{attribute 'pack_mode' := '1'}
TYPE ST_ReportListItem_Test :
STRUCT
    ReportType : STRING(50);
    ReportID   : STRING(50);
	CreatedOn  : STRING(30);
	CreatedBy  : STRING(50);
	Description : STRING(200);
	sPrimaryKey : STRING(50);
END_STRUCT
END_TYPE

(* stored: Version 1.1.0.1, ProductVersion 3.1.4024.15
   DUT ST_ReportListItem_Test: Id {b227047d-75e2-482b-8647-febf7e476446} *)
